TYPE ST_Empleado :
STRUCT
	Nombre 				: STRING;
    Apellido 			: STRING;
    CorreoElectronico 	: STRING;
END_STRUCT
END_TYPE

(* stored: Version 1.1.0.1, ProductVersion 3.1.4024.12
   DUT ST_Empleado: Id {70311c9f-0831-4fd9-b187-c603d6d25d14} *)
